RoboDK station: ejercicioRoboCuboLecturaTXT.rdk

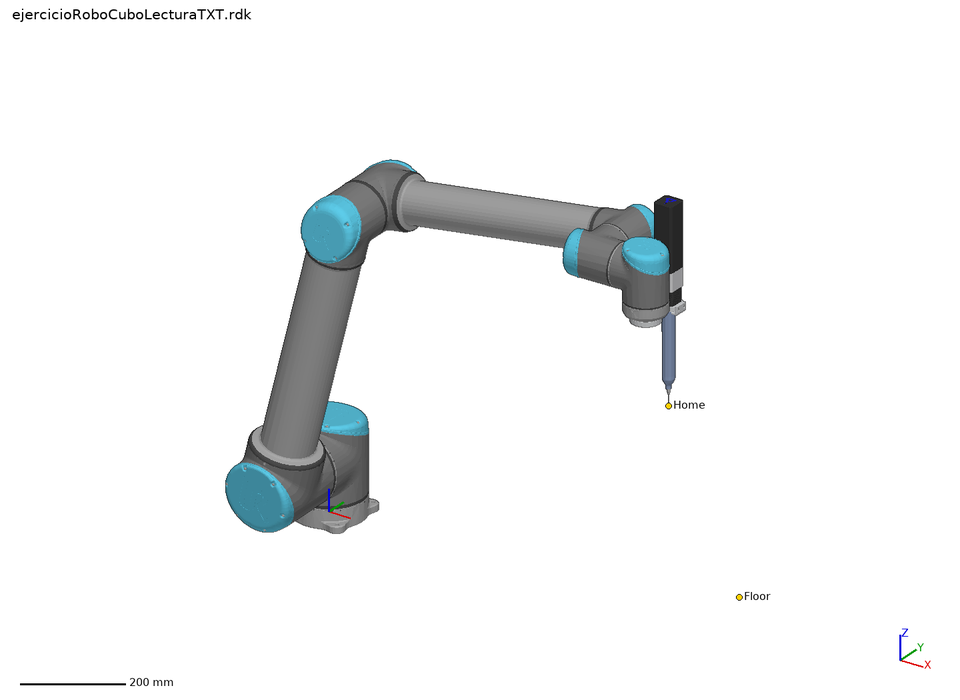
[picture v0: the station drawn from its stored meshes, robots at their saved joint values, targets as dots, program paths as lines]
Station ejercicioRoboCuboNew (saved by RoboDK 6.0.4). Poses are relative to the parent item; angles as X-Y-Z fixed-axis rotations.
  - frame UR10 Base at (2.24, 45.03, 606.3) mm
    - robot UR10: 6 axes, payload 10 kg, reach 1300 mm, repeatability 0.1 mm, weight 28.9 kg
        modified DH rows (alpha deg, a mm, theta deg, d mm): 0, 0, 0, 128; 90, 0, 180, 0; 0, 612.7, 0, 0; 0, 571.6, 0, 163.9; -90, 0, 0, 115.7; 90, 0, 180, 92.2
        joint limits [-360, -360, -360, -360, -360, -360] to [360, 360, 360, 360, 360, 360]; home [0, -90, -90, 0, 90, 0]; saved at [1.302, -103.964, -68.526, -97.51, 90, -88.698]
      - tool Dispenser , TCP at (0, -75, 221.24) mm, rotated rx 0 ry 0 rz 90 deg, size 63 x 128.2 x 432.2 mm
    - target Home (Cartesian target) at (833.75, -70, 483.87) mm, rotated rx 180 ry 0 rz -90 deg; joints [1.302, -103.964, -68.526, -97.51, 90, -88.698] of UR10
    - target Floor (Cartesian target) at (892.49, 80, 37.72) mm, rotated rx -179.06 ry 0 rz -90 deg; joints [10.966, -117.608, -96.64, -54.833, 89.822, -79.035] of UR10
  - Python program Cubo (listed below)
  - Python program EJ (listed below)

--- Python program Cubo ---
# Importamos Librerias
from robodk.robolink import *
from robodk.robomath import *

# Crear Instancia de la Clase RoboLink
rLink = Robolink()

# Obtenemos el Robot selecionado
Robot = rLink.Item('', ITEM_TYPE_ROBOT)

# Vincular variables de Python con targets
varHome = rLink.Item('Home')
varSuelo = rLink.Item('Floor')

# Comprovar el movimiento del robot.
Robot.MoveL(varHome)
Robot.MoveL(varSuelo)

# Obtener la Posicion de Referencia (Pose)
PosRef = varSuelo.Pose()

# Parametros del cubo
Lado = 200          # Tamaño del lado del cuadrado (mm). Subir este valor lo hace más amplio
Capas = 50          # Numero de capas apiladas
PasoAltura = -4     # Negativo para que suba hacia Home. 50 capas * 4 = 200 mm de alto (cubo)

# Esquinas de la base del cuadrado (en el plano del suelo)
Esquinas = [(0, 0), (Lado, 0), (Lado, Lado), (0, Lado)]

Eje_Z = 0
# Dibujar las capas cuadradas, subiendo en cada vuelta
for capa in range(Capas):
    # Recorrer el perimetro del cuadrado a la altura actual
    for x, y in Esquinas + [Esquinas[0]]:   # +primera esquina para cerrar
        Robot.MoveL(PosRef * transl(x, y, Eje_Z))
    # Subir a la siguiente capa
    Eje_Z = Eje_Z + PasoAltura

# Regresar a Home
Robot.MoveL(varHome)

--- Python program EJ ---
# Type help("robodk.robolink") or help("robodk.robomath") for more information
# Press F5 to run the script
# Documentation: https://robodk.com/doc/en/RoboDK-API.html
# Reference:     https://robodk.com/doc/en/PythonAPI/robodk.html
# Note: It is not required to keep a copy of this file, your Python script is saved with your RDK project

# You can also use the new version of the API:
from robodk import robolink    # RoboDK API
from robodk import robomath    # Robot toolbox

RDK = robolink.Robolink()

robot = RDK.Item('', robolink.ITEM_TYPE_ROBOT)

targetHome = RDK.Item('Home')
targetFloor = RDK.Item('Floor')

dato = ''

while dato != '0':
    with open('C:/Users/omar.fernandez/AppData/Local/Temp/ejRobodk.txt', 'r') as datoArchivo:
        dato = datoArchivo.readline().strip()
        print("Dato recibido: ", dato)
    match dato:
        case '1': robot.MoveJ(targetHome)
        case '2': robot.MoveJ(targetFloor)
